TEXTLIST AxesDialogAlphaUnitsTextList
  0 = 'h / m / s'
  1 = 'hours'
  2 = 'radians'
   = ''
END_TEXTLIST

(* stored: Version 1.1.0.1, ProductVersion 3.1.4018.5
   TextList AxesDialogAlphaUnitsTextList: Id {47466619-de99-4d95-b2e8-4237b09c8dd1} *)
